// Brief: Slave Arm test
FUNCTION_BLOCK PUBLIC FB_SlaveCtrlTest EXTENDS FB_SlaveArmCtrlBase
VAR_INPUT
END_VAR
VAR_OUTPUT
END_VAR
VAR
// ################ variables for single DH  joint test ##################
	m_enableFrictionComp :BOOL :=false;
	m_freqTestFlag :BOOL:=FALSE;
	m_initJntPos :Vec6d;
	m_cmdDHJntPos :Vec6d;
	m_cmdDHJntVel :Vec6d;
	m_cmdGripAng:LREAL;
	m_jntMotionFreq :Vec6d :=[0.2, 0.2, 0.1, 3(0.1)];
	m_jntMotionRange :Vec6d :=[pi/6, pi/6, 0.1, 3(pi/6)];
	m_testJntIdx :INT :=1;
	m_gripperAngle : LREAL :=0;
	m_gripForceLevel :LREAL :=0;
	m_lastCmdJntPos :Vec8d ;
	
	m_stepTestFlag :BOOL :=FALSE;
	m_jntStep : LREAL := 5*g_deg2Rad;
	
	// instrument controller
	m_instruController : FB_BasicInstruControl;
	m_usKnifeController : FB_UltrosonicKnifeControl;
	m_instruCmdJntPos,m_instruCmdJntVel : Vec5d;
	m_instruCmdJntTrq :Vec5d;
	m_maxGripCurrent:LREAL:=350.0;
	m_maxGripCtrlCurrent:LREAL:=540.0;
	
	m_errCmdPos, m_errCurPos :LREAL;
	m_errPosIdx : INT;
	
	m_originalJntPos:Vec8d;
		m_jntOTG:array[1..6] of FB_secOrdTrajFilter;
		m_gripAngleOTG : FB_secOrdTrajFilter;
	
//####################################################################

END_VAR

METHOD PROTECTED calcCmdJntPos : BOOL
VAR_IN_OUT CONSTANT
	i_endoscopePose : ST_Frame;
	i_masterStatus :ST_MasterStatus;
	i_setupStatus: ST_SetupStatus;
	i_slaveArm :FB_SlaveArm;
END_VAR

VAR 
	i:INT :=0;
	errThres :LREAL;

END_VAR
IF m_testJntIdx <4 OR m_testJntIdx >6 THEN
	RETURN;
END_IF

// frequency test
IF m_freqTestFlag THEN 
	m_cmdDHJntPos[m_testJntIdx]:=m_initJntPos[m_testJntIdx]+m_jntMotionRange[m_testJntIdx]/2
									+0.5*m_jntMotionRange[m_testJntIdx]*SIN(2*pi*m_jntMotionFreq[m_testJntIdx]*m_timePeriod-pi/2);
	m_cmdDHJntVel[m_testJntIdx]:=0.5*m_jntMotionRange[m_testJntIdx]*2*pi*m_jntMotionFreq[m_testJntIdx]*COS(2*pi*m_jntMotionFreq[m_testJntIdx]*m_timePeriod-pi/2);
// step test
ELSIF m_stepTestFlag THEN;
	m_jntOTG[m_testJntIdx].run(m_initJntPos[m_testJntIdx]+m_jntStep,0.0, o_cmdAcc=>,o_cmdVel=>m_cmdDHJntVel[m_testJntIdx],o_cmdPos=> m_cmdDHJntPos[m_testJntIdx]);
// reset controller
ELSE
	m_timePeriod:=0;
	m_initJntPos :=i_slaveArm.curDHJntPos;
	m_originalJntPos := i_slaveArm.curJntPos;
	m_cmdDHJntPos :=m_initJntPos;
	m_cmdDHJntVel :=g_zeroVec6d;
	m_gripperAngle := i_slaveArm.curGripAngle;
	// init instrument controller
	m_instruController.init(i_slaveArm,m_maxGripCurrent,m_maxGripCtrlCurrent);
	m_usKnifeController.init(i_slaveArm);
	
	FOR i:=1 TO 6  DO
		m_jntOTG[i].init(m_initJntPos[i], 0,12, 100, g_slaveArmCtrlCycleTime);
	END_FOR
	
	m_gripAngleOTG.init(m_gripperAngle, 0, 2, 8, g_slaveArmCtrlCycleTime);
END_IF

// calculate target motor joint position from DH joint position
m_gripAngleOTG.run(m_gripperAngle,0.0, o_cmdAcc=>,o_cmdVel=>,o_cmdPos=>m_cmdGripAng);
i_slaveArm.instrument.instruIK(m_cmdDHJntPos,m_cmdGripAng, o_jntPos=>m_cmdJntPos);

// command velocity
vecSub(m_cmdJntPos, m_lastCmdJntPos, m_cmdJntVel);
vecSelfMultiNum(m_cmdJntVel, g_slaveArmCtrlFreq);
m_lastCmdJntPos:=m_cmdJntPos;
END_METHOD

// override this function in each exact controller
METHOD PROTECTED calcCmdJntTrq : BOOL
VAR_IN_OUT CONSTANT
	i_endoscopePose : ST_Frame;
	i_masterStatus :ST_MasterStatus;
	i_setupStatus: ST_SetupStatus;
	i_slaveArm :FB_SlaveArm;
END_VAR

VAR 
	nullspaceMat :Mat7d;
	ctrlTrq : Vec7d;
	i : int ;
END_VAR
// set joint torque to zero in default
m_cmdJntTrq := g_zeroVec8d;

// instrument joint control
FOR i:=1 TO 5 DO 
	m_instruCmdJntPos[i]:=m_cmdJntPos[i+3];
	m_instruCmdJntVel[i]:=m_cmdJntVel[i+3];
END_FOR

IF i_slaveArm.instrument.instruType = InstruType_UltrasoundKnifeS OR i_slaveArm.instrument.instruType = InstruType_UltrasoundKnifeU THEN
	m_usKnifeController.run(m_instruCmdJntPos,m_instruCmdJntVel, m_gripForceLevel, i_slaveArm, o_cmdJntTrq=>m_instruCmdJntTrq);
ELSE
	m_instruController.run(m_instruCmdJntPos,m_instruCmdJntVel, m_cmdDHJntPos[6], m_cmdDHJntVel[6], m_gripForceLevel, i_slaveArm, o_cmdJntTrq=>m_instruCmdJntTrq);
END_IF

FOR i:=1 TO 5 DO
	m_cmdJntTrq[i+3]:=m_instruCmdJntTrq[i];
END_FOR

// add friction
IF m_enableFrictionComp THEN
	enableFrictionCompensation(i_slaveArm);
END_IF
END_METHOD

METHOD PUBLIC init : BOOL
VAR_IN_OUT CONSTANT
	i_slaveArm	:FB_SlaveArm;
END_VAR
VAR_IN_OUT 
	r_slaveArmCtrlCmd :ST_SlaveArmCtrlCmds;
END_VAR

VAR
	i:int;
END_VAR
SUPER^.Init(i_slaveArm,r_slaveArmCtrlCmd);
m_lastCmdJntPos:=m_cmdJntPos;
m_jntOPMode[1] := DriverOPMode_PosTrq;
m_jntOPMode[2] := DriverOPMode_PosTrq;
m_jntOPMode[3] := DriverOPMode_PosTrq;
m_jntOPMode[4] := DriverOPMode_Trq;
m_jntOPMode[5] := DriverOPMode_Trq;
m_jntOPMode[6] := DriverOPMode_Trq;
m_jntOPMode[7] := DriverOPMode_Trq;
m_jntOPMode[8] := DriverOPMode_Trq;

m_initJntPos :=i_slaveArm.curDHJntPos;
m_originalJntPos := i_slaveArm.curJntPos;
m_cmdDHJntPos :=m_initJntPos;
m_cmdDHJntVel :=g_zeroVec6d;
m_gripperAngle := i_slaveArm.curGripAngle;

// init instrument controller
m_instruController.init(i_slaveArm,m_maxGripCurrent,m_maxGripCtrlCurrent);
m_usKnifeController.init(i_slaveArm);

FOR i:=1 TO 6  DO
	m_jntOTG[i].init(m_initJntPos[i], 0,12, 100, g_slaveArmCtrlCycleTime);
END_FOR

m_gripAngleOTG.init(m_gripperAngle, 0,2, 8, g_slaveArmCtrlCycleTime);
// update commands to arm
copyCmds(r_slaveArmCtrlCmd);
END_METHOD

END_FUNCTION_BLOCK

(* stored: Version 1.1.0.1, ProductVersion 3.1.4024.11
   POU FB_SlaveCtrlTest: Id {25b7ca7b-a3c0-4d1d-9db6-09421c0085dc}, SpecialFunc None
   Method calcCmdJntPos: Id {010d1f8e-611a-45d6-a3e6-a98e946007a3}
   Method calcCmdJntTrq: Id {7ca43581-7589-4aef-a767-3681b3b7ea42}
   Method init: Id {59631f67-fc70-45f4-a6d2-b7e272ec8be8} *)
